Fanuc KAREL source: kd00060.KL

-- PROVISIONAL review KL for V770-1; original PC SHA256 746e32cc0ac48a884f015fdbf575e2d89a42487b745d09f5b0db3fc37fbaf0c2
-- Incomplete behavior may be omitted. Consult companion uncertainty JSON. Do not deploy.
PROGRAM KD00060
%NOLOCKGROUP
VAR
  I : INTEGER
  J : INTEGER
  B : BOOLEAN
  R : REAL
  S : STRING[80]
BEGIN
  -- UNRESOLVED_PC offsets 5-18; opcodes 9D,81,18,9D,1B,9D,12,9D,13,04
  -- UNRESOLVED_PC offsets 23-27; opcodes 7F
END KD00060
